FUNCTION_BLOCK LogBuffer
VAR_INPUT
END_VAR
VAR_OUTPUT
END_VAR
VAR
	logMessages : ARRAY [0..cMax] OF STRING(255);
	counter: INT := 0;
END_VAR
VAR CONSTANT
	cMax: INT := 100;
END_VAR

METHOD append : BOOL
VAR_INPUT
	message: STRING(255);
END_VAR
IF counter <= cMax
	THEN
	
	logMessages[counter] := message;
	counter := counter + 1;
	append := TRUE;
ELSE
	append := FALSE;
END_IF
END_METHOD

PROPERTY logAvailable : Bool
GET
logAvailable := (counter > 0);
END_GET
END_PROPERTY

METHOD pop : BOOL
VAR_IN_OUT
	message : STRING(255);
END_VAR
VAR
	popMessage: INT;
END_VAR
IF counter = 0 AND logMessages[counter] = ''
	THEN
	
	pop := FALSE;
	
ELSIF counter > 0
	THEN
	
	pop := TRUE;
	
	popMessage := counter - 1;
	message := logMessages[popMessage];
	logMessages[popMessage] := '';
	counter := popMessage;
	
END_IF
END_METHOD

END_FUNCTION_BLOCK

(* stored: Version 1.1.0.1, ProductVersion 3.1.4024.12
   POU LogBuffer: Id {24356b2b-138f-49d1-a985-3f05ee70eaf8}, SpecialFunc None
   Method append: Id {b2f9d90a-ce7c-42ef-baa1-b8377d686449}
   Property logAvailable: Id {5b1edc72-2d47-4151-82d5-fa9d4553d846}
   Get Get: Id {e32d3a85-798f-45fa-86f6-5158c542ea85}
   Method pop: Id {deb38650-8802-48cf-b795-a6ffaace8482} *)
